(* PLC project SafeLOGIC-1, BrAutomation SafeDESIGNER  4.4.0.0 *)
(* stored: companyURL http://www.br-automation.com, creationDateTime Mon Nov 08 10:35:14 2021 *)

PROGRAM Main
  VAR  (* added by the conversion: wires and edge detectors of the diagram *)
    _AND_S4_OUT : ANY;
    _SAFEBOOL_TO_BOOL34_OUT : BOOL;
  END_VAR

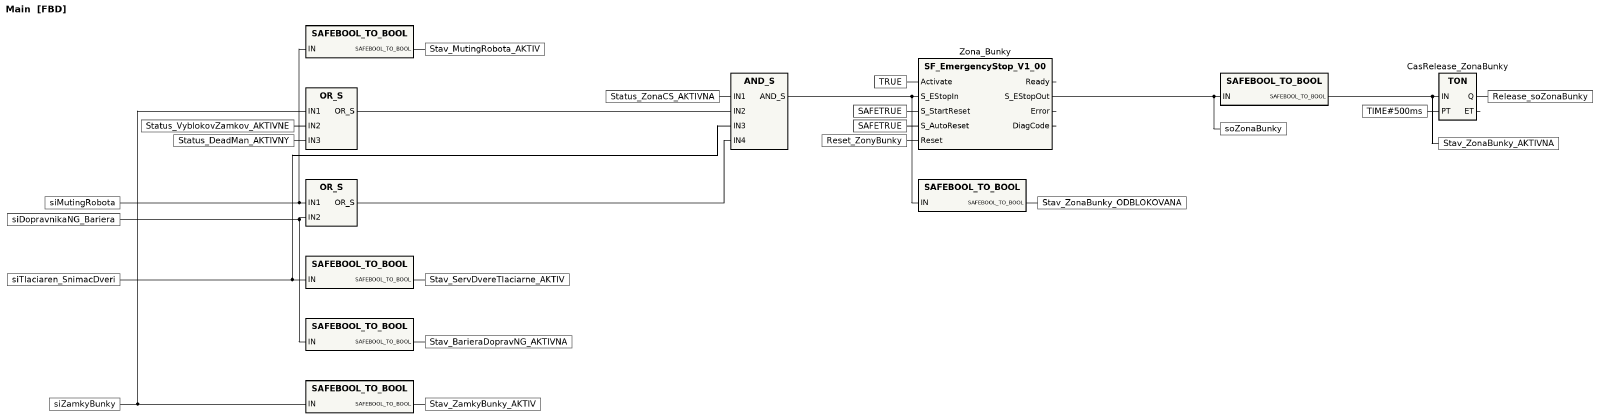
(* FBD diagram, written out as Structured Text *)
_AND_S4_OUT := AND_S(Status_ZonaCS_AKTIVNA, OR_S(siZamkyBunky, Status_VyblokovZamkov_AKTIVNE, Status_DeadMan_AKTIVNY), siTlaciaren_SnimacDveri, OR_S(siMutingRobota, siDopravnikaNG_Bariera));
Zona_Bunky(Activate := TRUE, S_EStopIn := _AND_S4_OUT, S_StartReset := SAFETRUE, S_AutoReset := SAFETRUE, Reset := Reset_ZonyBunky);
soZonaBunky := Zona_Bunky.S_EStopOut;
Stav_ZamkyBunky_AKTIV := SAFEBOOL_TO_BOOL(siZamkyBunky);
_SAFEBOOL_TO_BOOL34_OUT := SAFEBOOL_TO_BOOL(Zona_Bunky.S_EStopOut);
CasRelease_ZonaBunky(IN := _SAFEBOOL_TO_BOOL34_OUT, PT := TIME#500ms);
Release_soZonaBunky := CasRelease_ZonaBunky.Q;
Stav_ServDvereTlaciarne_AKTIV := SAFEBOOL_TO_BOOL(siTlaciaren_SnimacDveri);
Stav_ZonaBunky_ODBLOKOVANA := SAFEBOOL_TO_BOOL(_AND_S4_OUT);
Stav_ZonaBunky_AKTIVNA := _SAFEBOOL_TO_BOOL34_OUT;
Stav_MutingRobota_AKTIV := SAFEBOOL_TO_BOOL(siMutingRobota);
Stav_BarieraDopravNG_AKTIVNA := SAFEBOOL_TO_BOOL(siDopravnikaNG_Bariera);
END_PROGRAM
